// TIA Portal V19 export
FUNCTION_BLOCK "PN Port Status"   // FB5, LAD
{ S7_Optimized_Access := 'TRUE' }
// stored: MemoryReserve 100, SetENOAutomatically false
   VAR_INPUT
      HW_ID : HW_IO;
      Update : Bool;
   END_VAR
   VAR_OUTPUT
      Connected : Bool;
   END_VAR
   VAR
      Updated_ReqP : Bool;
      Updated_Req : Bool;
      RDREC_Instance { S7_SetPoint := 'True'} : RDREC;
   END_VAR
   VAR_TEMP
      Record : Struct
         BlockType : Word;
         BlockLength : UInt;
         BlockVersionHigh : USInt;
         BlockVersionLow : USInt;
         Padding : Word;
         SlotNumber : Word;
         SubSlotNumber : Word;
         Data : Array[0..299] of Byte;
      END_STRUCT;
      n : Array[0..3] of UInt;
      LinkState : Word;
   END_VAR
   VAR_TEMP   // added for the SCL form of the ladder/FBD networks
      _w1 : Bool;
   END_VAR
BEGIN

REGION Network 1: Positive Edge triggered Update Req
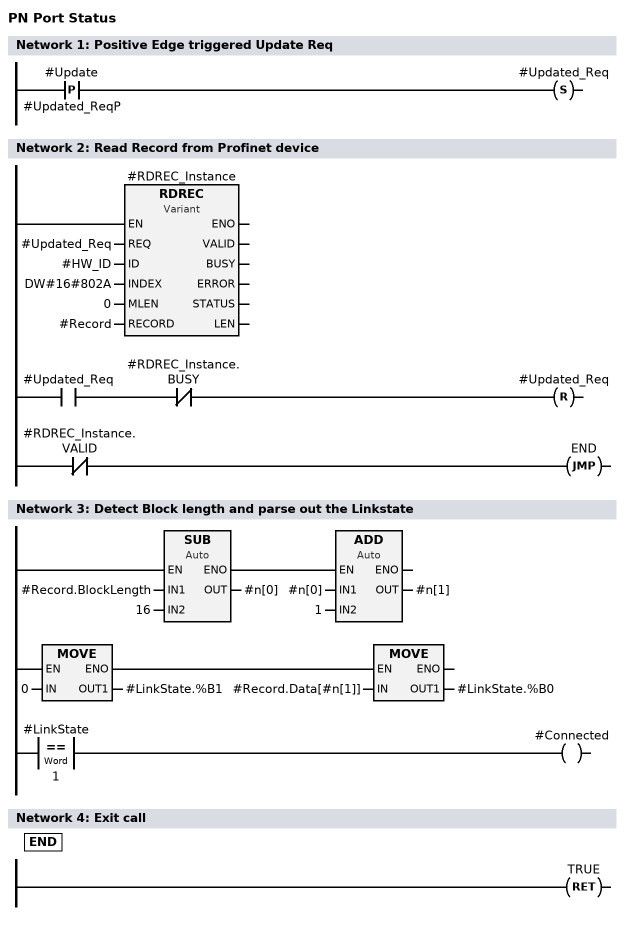
   RUNG wire#powerrail
      P_Contact(operand := #Update, bit := #Updated_ReqP)
      S_Coil( #Updated_Req )
   END_RUNG
   // the same network as SCL:
   #_w1 := #Update AND NOT #Updated_ReqP;   // rising edge of #Update
   #Updated_ReqP := #Update;
   IF #_w1 THEN #Updated_Req := TRUE; END_IF;
END_REGION

REGION Network 2: Read Record from Profinet device
   RUNG wire#powerrail
      { S7_Templates := "[ptr_type := Variant, id_type := HW_IO, index_type := DInt, len_type := UInt]" } #RDREC_Instance.RDREC(REQ := #Updated_Req, ID := #HW_ID, INDEX := DW#16#802A, MLEN := 0, RECORD := #Record, VALID =>, BUSY =>, ERROR =>, STATUS =>, LEN =>)
   END_RUNG
   RUNG wire#powerrail
      Contact( #Updated_Req )
      I_Contact( #RDREC_Instance.BUSY )
      R_Coil( #Updated_Req )
   END_RUNG
   RUNG wire#powerrail
      I_Contact( #RDREC_Instance.VALID )
      JumpCoil( END )
   END_RUNG
   // the same network as SCL:
   #RDREC_Instance(REQ := #Updated_Req, ID := #HW_ID, INDEX := DW#16#802A, MLEN := 0, RECORD := #Record);   // RDREC
   IF #Updated_Req AND NOT #RDREC_Instance.BUSY THEN #Updated_Req := FALSE; END_IF;
   IF NOT #RDREC_Instance.VALID THEN GOTO END; END_IF;
END_REGION

REGION Network 3: Detect Block length and parse out the Linkstate
   RUNG wire#powerrail
      Sub(in1 := #Record.BlockLength, in2 := 16, out => #n[0])
      Add(in1 := #n[0], in2 := 1, out => #n[1])
   END_RUNG
   RUNG wire#powerrail
      Move(in := 0, out1 => #LinkState.%B1)
      Move(in := #Record.Data[#n[1]], out1 => #LinkState.%B0)
   END_RUNG
   RUNG wire#powerrail
      { S7_Templates := "SrcType := Word" } EQ_Contact(in1 := #LinkState, in2 := 1)
      Coil( #Connected )
   END_RUNG
   // the same network as SCL:
   #n[0] := #Record.BlockLength - 16;
   #n[1] := #n[0] + 1;
   #LinkState.%B1 := 0;
   #LinkState.%B0 := #Record.Data[#n[1]];
   #Connected := #LinkState = 1;
END_REGION

REGION Network 4: Exit call
   END:
   ENO := TRUE;
   RETURN;
END_REGION
END_FUNCTION_BLOCK
